FUNCTION_BLOCK fb_prod_rate

VAR_INPUT
	set_prod_rate: REAL;
	xmv17: REAL;
	kc: REAL;
	ti:REAL;
	ts:REAL;
	hi:REAL;
	lo:REAL;
	x0:REAL;
END_VAR

VAR_OUTPUT
	Prodsp: REAL;
	Fp: REAL;
END_VAR

VAR
	vel_p: fb_vel_pi;
	x: FB_CTRL_2POINT;
	zoh_real_0: fb_zoh_real := (last := x0);
	change_rate_limit: FB_CTRL_LIMITER := (stInternalParams := (fMinOutput := -0.3, fMaxOutput := 0.3));
	rate: REAL := 0;
	ProdspGain: REAL := 100/22.89;
	prodsp_scaled: REAL;
	calc_change_rate: FB_CTRL_D;
	integrate_change_rate: FB_CTRL_I;
	prod_rate_saturate: FB_CTRL_LIMITER;
	prod_rate_saturate_params: ST_CTRL_LIMITER_PARAMS := (fMinOutput := lo, fMaxOutput := hi);
	last_prod_rate: REAL := 0.0;
	
	stparams_calc_change_rate: ST_CTRL_D_PARAMS;
	stparams_change_rate_limit: ST_CTRL_LIMITER_PARAMS;
	stparams_integrate_change_rate: ST_CTRL_I_PARAMS;
	
END_VAR

VAR CONSTANT

END_VAR

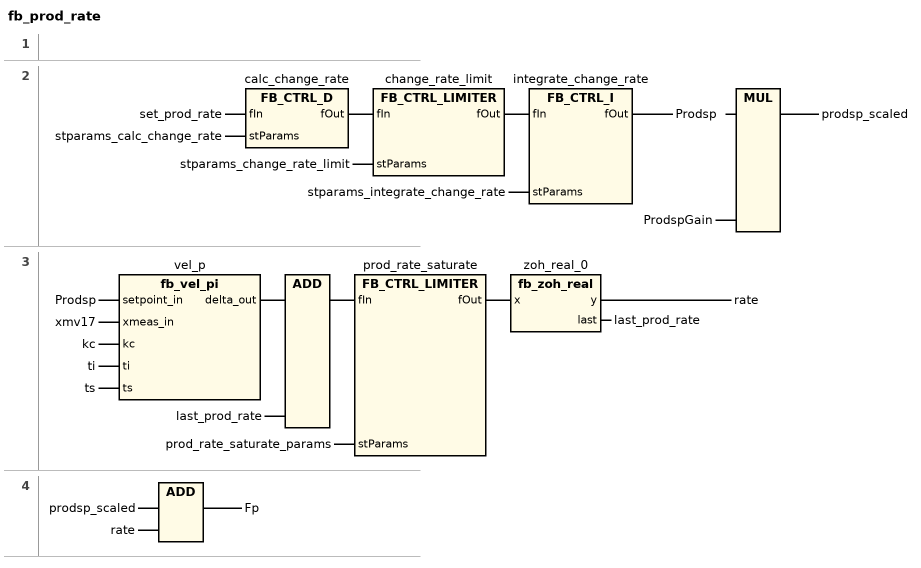
// NETWORK 1

// NETWORK 2
calc_change_rate(fIn := set_prod_rate, stParams := stparams_calc_change_rate); // FB_CTRL_D
change_rate_limit(fIn := calc_change_rate.fOut, stParams := stparams_change_rate_limit); // FB_CTRL_LIMITER
integrate_change_rate(fIn := change_rate_limit.fOut, stParams := stparams_integrate_change_rate); // FB_CTRL_I
Prodsp := integrate_change_rate.fOut;
prodsp_scaled := integrate_change_rate.fOut * ProdspGain;

// NETWORK 3
vel_p(setpoint_in := Prodsp, xmeas_in := xmv17, kc := kc, ti := ti, ts := ts); // fb_vel_pi
prod_rate_saturate(fIn := vel_p.delta_out + last_prod_rate, stParams := prod_rate_saturate_params); // FB_CTRL_LIMITER
zoh_real_0(x := prod_rate_saturate.fOut, last => last_prod_rate); // fb_zoh_real
rate := zoh_real_0.y;

// NETWORK 4
Fp := prodsp_scaled + rate;

END_FUNCTION_BLOCK

(* stored: Version 1.1.0.1, ProductVersion 3.1.0.26
   POU fb_prod_rate: Id {12afc640-1cc9-456e-b128-0a54a95b7ca0} *)
